FUNCTION_BLOCK COLOR_POS_RED (* Basic Function Block Type *)
  (* Standard: 61499-2 *)
  (* Version 0.3, 2009-09-15, JHC, Holobloc Inc, Changed transition priorities. *)
  (* Version 0.2, 2003-12-04, JHC, Rockwell Automation, Renamed for better indexing. *)
  (* Version 0.1, 2002-11-05, JHC, Rockwell Automation, Corrected missing ST element in Algorithm REQ. *)
  (* Version 0.0, 2000-05-30, JHC, Rockwell Automation *)
  PACKAGE fb.rt.Conveyer;
  IMPORT fb.datatype.*;
  IMPORT fb.rt.*;
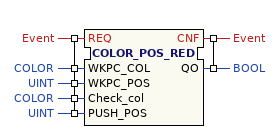
  EVENT_INPUT
    REQ WITH WKPC_COL, WKPC_POS, Check_col, PUSH_POS; (* Normal Execution Request *)
  END_EVENT
  EVENT_OUTPUT
    CNF WITH QO; (* Execution Confirmation *)
  END_EVENT
  VAR_INPUT
    WKPC_COL : COLOR;
    WKPC_POS : UINT;
    Check_col : COLOR;
    PUSH_POS : UINT;
  END_VAR
  VAR_OUTPUT
    QO : BOOL; (* Output event qualifier *)
  END_VAR
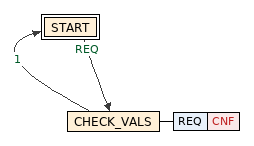
  EC_STATES
    START; (* Initial State *)
    CHECK_VALS : REQ -> CNF; (* Normal execution *)
  END_STATES
  EC_TRANSITIONS
    START TO CHECK_VALS := REQ;
    CHECK_VALS TO START := 1;
  END_TRANSITIONS
  ALGORITHM REQ IN ST: (* Normally executed algorithm *)
IF  (WKPC_POS>=PUSH_POS) THEN
	QO := FALSE;
ELSE
	QO := FALSE;
END_IF;

IF (WKPC_COL=Check_col) THEN
	QO := TRUE;
END_IF;
  END_ALGORITHM
END_FUNCTION_BLOCK
